(* IEC 61131-3 sources: GradProject/PLC/LadderLogic, 2 files *)

(* ---- Test23.st ---- *)
PROGRAM Test_Program
  VAR
    ESP0 AT %QX0.0 : BOOL;
  END_VAR
  VAR
    TMP : BOOL;
  END_VAR
  VAR
    ESP1 AT %QX0.1 : BOOL;
  END_VAR
  VAR
    TON1 : TON;
    TON2 : TON;
  END_VAR

  IF NOT(TMP) THEN
    ESP0 := TRUE; (*set*)
  END_IF;
  TON1(IN := ESP0, PT := T#10000ms);
  IF TON1.Q THEN
    ESP1 := TRUE; (*set*)
  END_IF;
  TON2(IN := ESP1, PT := T#10000ms);
  IF TON2.Q THEN
    ESP1 := FALSE; (*reset*)
  END_IF;
  IF TON2.Q THEN
    ESP0 := FALSE; (*reset*)
  END_IF;
END_PROGRAM

CONFIGURATION Config0

  RESOURCE Res0 ON PLC
    TASK MyTask(INTERVAL := T#50ms,PRIORITY := 0);
    PROGRAM instance0 WITH MyTask : Test_Program;
  END_RESOURCE
END_CONFIGURATION

(* ---- Test27.st ---- *)
PROGRAM Test_Program
  VAR
    ESP0 AT %QX0.0 : BOOL;
    TMP AT %QX0.2 : BOOL;
    ESP1 AT %QX0.1 : BOOL;
  END_VAR
  VAR
    TON1 : TON;
    TON2 : TON;
  END_VAR

  TMP := TRUE;
  ESP0 := TRUE;
  TON1(IN := ESP0 OR ESP0, PT := T#3000ms);
  ESP1 := TON1.Q;
  TON2(IN := ESP1, PT := T#5000ms);
  TMP := TON2.Q;
END_PROGRAM

CONFIGURATION Config0

  RESOURCE Res0 ON PLC
    TASK MyTask(INTERVAL := T#50ms,PRIORITY := 0);
    PROGRAM instance0 WITH MyTask : Test_Program;
  END_RESOURCE
END_CONFIGURATION
